SUBAPPLICATION Uebung_080f (* Beispiel für E_CTU *)
  (* Standard: 61499-2; Description: Copyright (c) 2023 Meisterschulen am Ostbahnhof This program and the accompanying materials are made available under the terms of the Eclipse Public License 2.0 which is available at https://www.eclipse.org/legal/epl-2.0/ SPDX-License-Identifier: EPL-2.0 *)
  (* Version 1.0, 2023-10-23, Franz Höpfinger, Meisterschulen am Ostbahnhof, initial API and implementation and/or initial documentation *)
  PACKAGE Uebungen;
  IMPORT Uebungen::const::UT::Horse::DefaultPool_Horse::ObjectPointer_Horse;
  IMPORT Uebungen::const::UT::Horse::DefaultPool_Horse::frame_00;
  IMPORT Uebungen::const::UT::Horse::DefaultPool_Horse::frame_01;
  IMPORT Uebungen::const::UT::Horse::DefaultPool_Horse::frame_02;
  IMPORT Uebungen::const::UT::Horse::DefaultPool_Horse::frame_03;
  IMPORT Uebungen::const::UT::Horse::DefaultPool_Horse::frame_04;
  IMPORT Uebungen::const::UT::Horse::DefaultPool_Horse::frame_05;
  IMPORT Uebungen::const::UT::Horse::DefaultPool_Horse::frame_06;
  IMPORT Uebungen::const::UT::Horse::DefaultPool_Horse::frame_07;
  IMPORT Uebungen::const::UT::Horse::DefaultPool_Horse::frame_08;
  IMPORT Uebungen::const::UT::Horse::DefaultPool_Horse::frame_09;
  IMPORT Uebungen::const::UT::Horse::DefaultPool_Horse::frame_10;
  IMPORT Uebungen::const::UT::Horse::DefaultPool_Horse::frame_11;
  IMPORT Uebungen::const::UT::Horse::DefaultPool_Horse::frame_12;
  IMPORT Uebungen::const::UT::Horse::DefaultPool_Horse::frame_13;
  IMPORT Uebungen::const::UT::Horse::DefaultPool_Horse::frame_14;
  IMPORT Uebungen::const::UT::Horse::DefaultPool_Horse::frame_15;
  IMPORT Uebungen::const::UT::Horse::DefaultPool_Horse::frame_16;
  IMPORT Uebungen::const::UT::Horse::DefaultPool_Horse::frame_17;
  IMPORT Uebungen::const::UT::Horse::DefaultPool_Horse::frame_18;
  IMPORT Uebungen::const::UT::Horse::DefaultPool_Horse::frame_19;
  IMPORT Uebungen::const::UT::Horse::DefaultPool_Horse::frame_20;
  IMPORT Uebungen::const::UT::Horse::DefaultPool_Horse::frame_21;
  IMPORT Uebungen::const::UT::Horse::DefaultPool_Horse::frame_22;
  IMPORT Uebungen::const::UT::Horse::DefaultPool_Horse::frame_23;
  IMPORT Uebungen::const::UT::Horse::DefaultPool_Horse::frame_24;
  IMPORT Uebungen::const::UT::Horse::DefaultPool_Horse::frame_25;
  IMPORT Uebungen::const::UT::Horse::DefaultPool_Horse::frame_26;
  IMPORT Uebungen::const::UT::Horse::DefaultPool_Horse::frame_27;
  IMPORT Uebungen::const::UT::Horse::DefaultPool_Horse::frame_28;
  IMPORT Uebungen::const::UT::Horse::DefaultPool_Horse::frame_29;
  IMPORT Uebungen::const::UT::Horse::DefaultPool_Horse::frame_30;
  IMPORT Uebungen::const::UT::Horse::DefaultPool_Horse::frame_31;
  IMPORT logiBUS::io::DI::logiBUS_DI::Input_I1;
  IMPORT logiBUS::io::DI::logiBUS_DI::Input_I2;
  IMPORT logiBUS::io::DI::logiBUS_DI_Events::BUTTON_SINGLE_CLICK;
  IMPORT logiBUS::io::DQ::logiBUS_DO::Output_Q1;
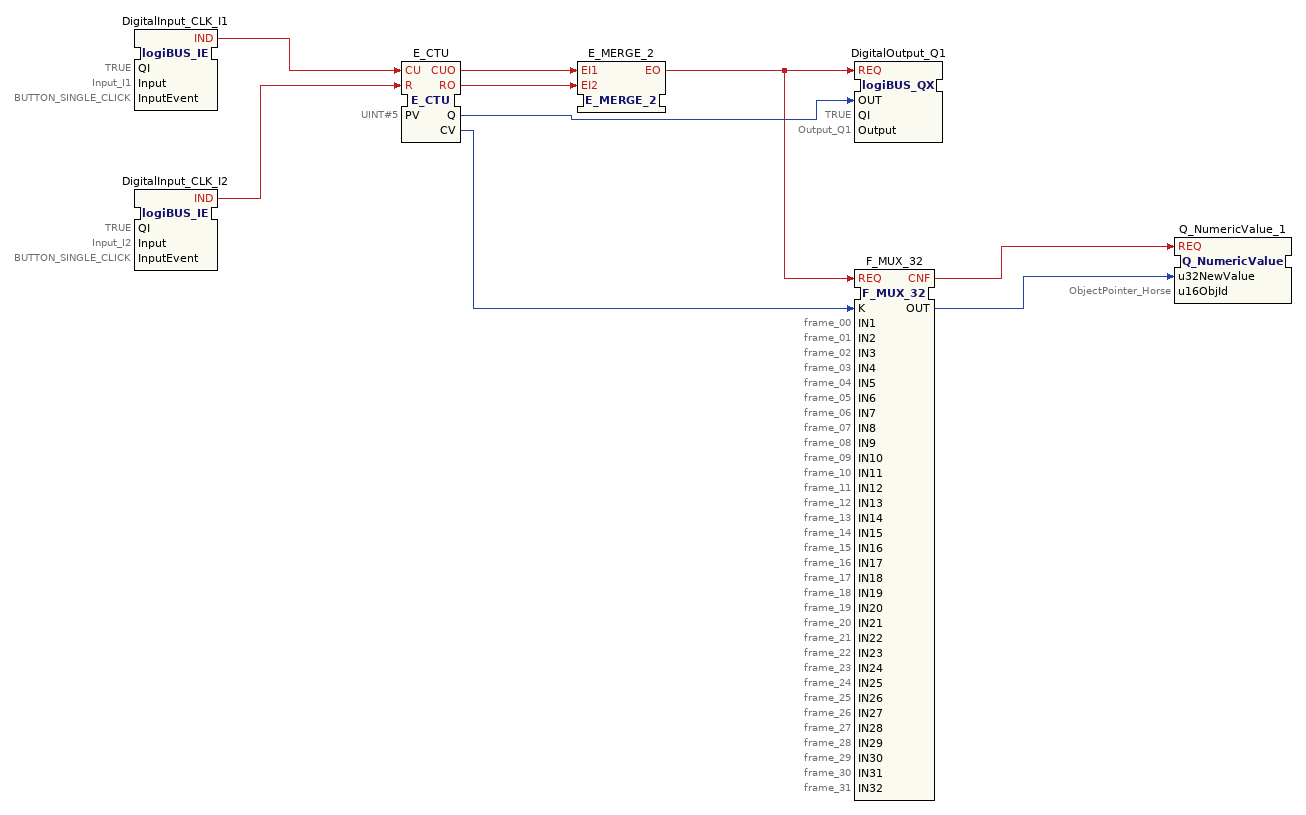
  (* da UDINT immer einen UINT aufnehmen kann, ist hier der UINT_TO_UDINT verzichtbar *)
  (* E_MERGE kann man weglassen, führt hier aber zu viel saubererem Code. (sonst muss man 4 Linien kreuzen) *)
  FBS
    DigitalOutput_Q1 : logiBUS::io::DQ::logiBUS_QX(QI := TRUE, Output := Output_Q1);
    DigitalInput_CLK_I1 : logiBUS::io::DI::logiBUS_IE(QI := TRUE, Input := Input_I1, InputEvent := BUTTON_SINGLE_CLICK);
    E_CTU : iec61499::events::E_CTU(PV := UINT#5);
    DigitalInput_CLK_I2 : logiBUS::io::DI::logiBUS_IE(QI := TRUE, Input := Input_I2, InputEvent := BUTTON_SINGLE_CLICK);
    E_MERGE_2 : iec61499::events::E_MERGE_2;
    Q_NumericValue_1 : isobus::UT::Q::Q_NumericValue(u16ObjId := ObjectPointer_Horse);
    F_MUX_32 : iec61131::selection::F_MUX_32(IN1 := frame_00, IN2 := frame_01, IN3 := frame_02, IN4 := frame_03, IN5 := frame_04, IN6 := frame_05, IN7 := frame_06, IN8 := frame_07, IN9 := frame_08, IN10 := frame_09, IN11 := frame_10, IN12 := frame_11, IN13 := frame_12, IN14 := frame_13, IN15 := frame_14, IN16 := frame_15, IN17 := frame_16, IN18 := frame_17, IN19 := frame_18, IN20 := frame_19, IN21 := frame_20, IN22 := frame_21, IN23 := frame_22, IN24 := frame_23, IN25 := frame_24, IN26 := frame_25, IN27 := frame_26, IN28 := frame_27, IN29 := frame_28, IN30 := frame_29, IN31 := frame_30, IN32 := frame_31);
  END_FBS
  EVENT_CONNECTIONS
    DigitalInput_CLK_I1.IND TO E_CTU.CU;
    DigitalInput_CLK_I2.IND TO E_CTU.R;
    E_CTU.CUO TO E_MERGE_2.EI1;
    E_CTU.RO TO E_MERGE_2.EI2;
    E_MERGE_2.EO TO DigitalOutput_Q1.REQ;
    F_MUX_32.CNF TO Q_NumericValue_1.REQ;
    E_MERGE_2.EO TO F_MUX_32.REQ;
  END_CONNECTIONS
  DATA_CONNECTIONS
    E_CTU.Q TO DigitalOutput_Q1.OUT;
    F_MUX_32.OUT TO Q_NumericValue_1.u32NewValue;
    E_CTU.CV TO F_MUX_32.K;
  END_CONNECTIONS
END_SUBAPPLICATION
